// TwinCAT 3 PLC project Main
// ProgramVersion: 3.1.4023.0
// libraries:
//   Tc2_Standard, * (Beckhoff Automation GmbH)
//   Tc2_System, * (Beckhoff Automation GmbH)
//   Tc3_JsonXml, * (Beckhoff Automation GmbH)
//   Tc3_Module, * (Beckhoff Automation GmbH)
// project tree:
//   Lib/QueueNode/ I_QueueNode.TcIO, QueueNode.TcPOU
//   Lib/Queue/ Queue.TcPOU
//   / PlcTask.TcTTO
//   POUs/ MAIN.TcPOU, Coordinate3D.TcDUT
// real-time tasks:
//   TASK PlcTask: cycle T#10ms, priority 20, ADS port 350

CONFIGURATION Main
    RESOURCE PLC ON TwinCAT3
        TASK PlcTask(INTERVAL := T#10ms, PRIORITY := 20);
        PROGRAM MAIN WITH PlcTask : MAIN;
    END_RESOURCE
END_CONFIGURATION

// ---- POUs/Coordinate3D.TcDUT
TYPE Coordinate3D :
STRUCT
	x : INT;
	y : INT;
	z : INT;
END_STRUCT
END_TYPE

// ---- Lib/QueueNode/I_QueueNode.TcIO
INTERFACE I_QueueNode

PROPERTY PUBLIC DataType : T_MaxString
GET
END_GET
END_PROPERTY

METHOD PUBLIC Destroy
VAR_INPUT
END_VAR
END_METHOD

METHOD PUBLIC Get : BOOL;
VAR_INPUT
	Destination : ANY;
END_VAR
END_METHOD

PROPERTY PUBLIC Next : I_QueueNode
GET
END_GET
SET
END_SET
END_PROPERTY

END_INTERFACE

// ---- POUs/MAIN.TcPOU
PROGRAM MAIN
VAR
	
	queue : Queue;
	size : UINT;
	
	// showing the use of the queue for the same datatype
	trigger : BOOL;
	position1 : Coordinate3D :=  (x:=3, y:=8, z:=-1);
	position2 : Coordinate3D :=  (x:=9, y:=1, z:=0);
	currentPosition : Coordinate3D;
	
	// showing the same queue can be used for anything at any time!
	trigger2 : BOOL;	
	myInt : INT := 123;
	myBool : BOOL := TRUE;
	myPosition : Coordinate3D :=  (x:=3, y:=8, z:=-1);
	poppedInt : INT;
	poppedBool : BOOL;
	poppedPosition : Coordinate3D;	
	
END_VAR

// example showing the queue can hold any number of the same type. 
IF trigger THEN
	
	trigger := FALSE;
	
	queue.Push(position1);
	queue.Push(position2);
	
	size := queue.Size(); // size 2
	queue.Pop(currentPosition); // (x:=3, y:=8, z:=-1)
	size := queue.Size(); // size 1
	queue.Pop(currentPosition); // (x:=9, y:=1, z:=0)
	size := queue.Size(); // size 0

END_IF

// example showing the queue can hold any number of any type all at the same time. 
IF trigger2 THEN
	
	trigger2 := FALSE;
	
	queue.Push(myInt);
	queue.Push(myBool);
	queue.Push(myPosition);
	
	size := queue.Size(); // size 3
	queue.Pop(poppedBool); // The datatype is wrong as the first push was an INT so nothing is popped.
	
	size := queue.Size(); // size 3
	queue.Pop(poppedInt); // 123
	size := queue.Size(); // size 2
	queue.Pop(poppedBool); // true
	size := queue.Size(); // size 1
	queue.Pop(poppedPosition); // (x:=3, y:=8, z:=-1)
	size := queue.Size(); // size 0
	
END_IF

END_PROGRAM

// ---- Lib/Queue/Queue.TcPOU
{attribute 'linkalways'}
{attribute 'no_explicit_call' := 'do not call this POU directly'}
FUNCTION_BLOCK Queue
VAR
	head : I_QueueNode;
END_VAR

METHOD PUBLIC Clear
VAR_INPUT
END_VAR
VAR
	current, next : I_QueueNode;
END_VAR
IF head = 0 THEN	
	RETURN;
END_IF

current := head; 

WHILE current.Next <> 0 DO
	next := current.next; 
	current.Destroy();
	current := next;
END_WHILE;
	
current.Destroy();
END_METHOD

METHOD FB_exit : BOOL
VAR_INPUT
	bInCopyCode : BOOL; // if TRUE, the exit method is called for exiting an instance that is copied afterwards (online change).
END_VAR
IF bInCopyCode THEN
	RETURN;
END_IF

Clear();
END_METHOD

METHOD PUBLIC Pop : BOOL;
VAR_INPUT
	Destination : ANY;
END_VAR
VAR
	transform : FB_JsonReadWriteDataType;
	next : I_QueueNode;
END_VAR
IF head = 0 THEN
	RETURN;
END_IF

IF head.DataType <> transform.GetDataTypeNameByAddress(Destination.diSize,Destination.pValue) THEN
	RETURN;
END_IF

next := head.Next;

Pop := head.Get(Destination);
head.Destroy();
head := next;
END_METHOD

METHOD PUBLIC Push
VAR_INPUT
	Item : ANY;
END_VAR
VAR
	pQueueNode : POINTER TO QueueNode;
	last : I_QueueNode;
END_VAR
pQueueNode := __NEW(QueueNode(Source := Item)); 

IF head = 0 THEN	
	head := pQueueNode^; 
	RETURN;
END_IF

last := head; 

WHILE last.Next <> 0 DO
	last := last.next; 
END_WHILE;
	
last.next := pQueueNode^;
END_METHOD

METHOD PUBLIC Size : UINT
VAR
	currentCount : UINT;
	currentNode : I_QueueNode;
END_VAR
currentCount := 0;
currentNode := head;

WHILE currentNode <> 0 DO
	currentNode := currentNode.Next;
	currentCount := currentCount + 1;
END_WHILE;

Size := currentCount;
END_METHOD

END_FUNCTION_BLOCK

// ---- Lib/QueueNode/QueueNode.TcPOU
{attribute 'linkalways'}
{attribute 'no_explicit_call' := 'do not call this POU directly'}
{attribute 'enable_dynamic_creation'}
FUNCTION_BLOCK QueueNode IMPLEMENTS I_QueueNode
VAR
	internalBuffer : POINTER TO BYTE;
	internalBufferSize : UDINT;
	sourceDataType : T_MAXSTRING;
	nextNode : I_QueueNode;
END_VAR

METHOD PRIVATE CopyInternalBufferToDestination
VAR_INPUT
	DestinationAddress : PVOID;
END_VAR
memcpy(DestinationAddress,internalBuffer,internalBufferSize);
END_METHOD

METHOD PRIVATE CopySourceToInternalBuffer
VAR_INPUT
	SourceAddress : PVOID;
END_VAR
memcpy(internalBuffer,SourceAddress,internalBufferSize);
END_METHOD

PROPERTY PUBLIC DataType : T_MaxString
GET
DataType := sourceDataType;
END_GET
END_PROPERTY

METHOD PRIVATE DeleteInternalBuffer
IF internalBuffer <> 0 THEN
	__DELETE(internalBuffer);
END_IF
END_METHOD

METHOD PUBLIC Destroy
VAR_INPUT
END_VAR
DeleteInternalBuffer();
__Delete(this);
END_METHOD

METHOD FB_init : BOOL
VAR_INPUT
	bInitRetains : BOOL; // if TRUE, the retain variables are initialized (warm start / cold start)
	bInCopyCode : BOOL;  // if TRUE, the instance afterwards gets moved into the copy code (online change)
	Source : ANY;
END_VAR
VAR
	transform : FB_JsonReadWriteDataType;
END_VAR
MakeInternalBufferOfSize(DINT_TO_UDINT(Source.diSize));
CopySourceToInternalBuffer(Source.pValue);
sourceDataType := transform.GetDataTypeNameByAddress(Source.diSize,Source.pValue);
END_METHOD

METHOD PUBLIC Get : BOOL;
VAR_INPUT
	Destination : ANY;
END_VAR
IF NOT IsInternalBufferSameSizeAs(DINT_TO_UDINT(Destination.diSize)) THEN
	RETURN;
END_IF

CopyInternalBufferToDestination(Destination.pValue);
END_METHOD

METHOD PRIVATE IsInternalBufferSameSizeAs : BOOL
VAR_INPUT
	Size : UDINT;
END_VAR
IF internalBuffer = 0 THEN
	RETURN;
END_IF

IF internalBufferSize <> Size THEN
	RETURN;
END_IF

IsInternalBufferSameSizeAs := TRUE;
END_METHOD

METHOD PRIVATE MakeInternalBufferOfSize
VAR_INPUT
	Size : UDINT;
END_VAR
internalBufferSize := Size;
internalBuffer := __NEW(BYTE, internalBufferSize);
END_METHOD

PROPERTY PUBLIC Next : I_QueueNode
GET
Next := nextNode;
END_GET
SET // PUBLIC
nextNode := Next;
END_SET
END_PROPERTY

END_FUNCTION_BLOCK
